FUNCTION_BLOCK E_DELAY (* Delayed propagation of an event (synthetic test fixture) *)
  PACKAGE IEC61499.Standard;
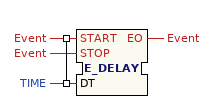
  EVENT_INPUT
    START WITH DT;
    STOP;
  END_EVENT
  EVENT_OUTPUT
    EO;
  END_EVENT
  VAR_INPUT
    DT : TIME;
  END_VAR
END_FUNCTION_BLOCK
